// Mitsubishi GX Works2 project: Pract02_Enclavamiento   PLC: FX3U/FX3UC

PROGRAM MAIN
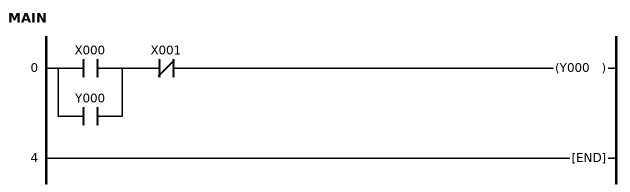
0     LD      X000
      OR      Y000
      ANI     X001
      OUT     Y000
4     END
END_PROGRAM
